FUNCTION "ST10_Analog" : Void
VAR_INPUT
  iSysMode : "RCS_SysComInterface_V1";
END_VAR
VAR_TEMP
  idex : Int;
END_VAR
BEGIN
  // Původní jazyk: SCL
  // Zdroj XML: EXPORT/Program blocks/OP010/10_Device/08_PressureAanlog/ST10_Analog.xml
  // --- Rekonstruovaný StructuredText (best-effort) ---
  // Network 1
  REGION

      #idex := ;

   END_REGION
END_FUNCTION
